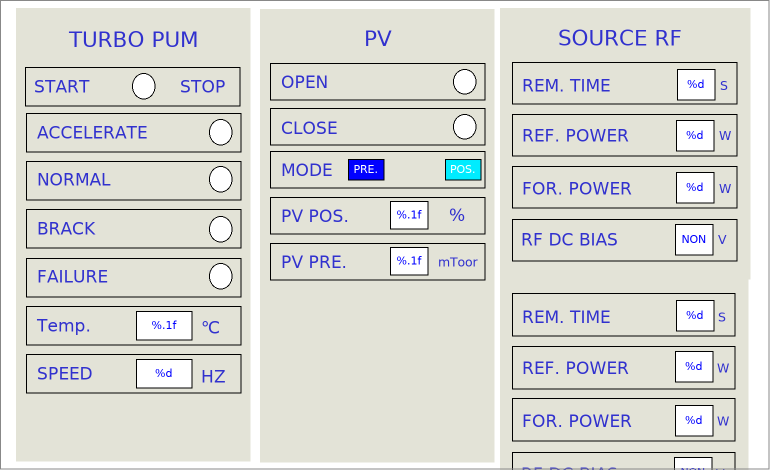
VISUALIZATION ViewPar  // 770x470
    RoundedRectangle (16,8 234x453)
    Label (38,17 192x45), "TURBO PUM"
    Ellipse (132,73 23x26), colour toggle: gICP.TruboPumOpen
    Label (31,75 67x23), "START"
    RoundedRectangle (26,113 215x39)
    RoundedRectangle (26,209 215x39)
    Ellipse (209,166 23x26), colour toggle: gICP.TruboPumNormal
    Label (34,168 117x23), "NORMAL"
    RoundedRectangle (26,161 215x39)
    Ellipse (209,119 23x26), colour toggle: gICP.TruboPumAcc
    Label (34,121 140x23), "ACCELERATE"
    RoundedRectangle (26,258 215x39)
    Ellipse (209,216 23x26), colour toggle: gICP.TruboPumDcc
    Label (34,217 117x23), "BRACK"
    RoundedRectangle (26,306 215x39)
    Ellipse (209,263 23x26), colour toggle: gICP.TruboPumError
    Label (34,265 117x23), "FAILURE"
    RoundedRectangle (26,354 215x39)
    Label (34,362 70x23), "SPEED"
    Label (198,365 31x23), "HZ"
    RoundedRectangle (136,359 56x29), "%d", text variable: gICP.TruboPumRotationSpeed
    Label (177,75 57x23), "STOP"
    Label (34,314 105x23), "Temp."
    Label (198,316 31x23), "℃"
    RoundedRectangle (136,311 56x29), "%.1f", text variable: gICP.TruboPumTMS
    RoundedRectangle (25,67 215x39)
    RoundedRectangle (260,9 234x453)
    Label (282,17 192x43), "PV"
    RoundedRectangle (270,63 215x37)
    Ellipse (453,69 23x25), colour toggle: gICP.PDVOpenSensor
    Label (278,71 117x22), "OPEN"
    RoundedRectangle (270,108 215x37)
    Ellipse (453,114 23x25), colour toggle: gICP.PDVCloseSensor
    Label (278,117 117x22), "CLOSE"
    RoundedRectangle (270,151 215x37)
    Label (278,159 69x22), "MODE"
    RoundedRectangle (270,197 215x37)
    Label (278,205 87x22), "PV POS."
    RoundedRectangle (270,243 215x37)
    Label (278,251 87x22), "PV PRE."
    RoundedRectangle (348,159 36x21), "PRE.", colour toggle: gICP.PDVModeRelay
    RoundedRectangle (445,159 36x21), "POS.", colour toggle: gICP.PDVModeRelay
    Label (446,204 23x22), "%"
    RoundedRectangle (390,201 38x28), "%.1f", text variable: gICP.PDV.actPos
    RoundedRectangle (390,247 38x28), "%.1f", text variable: gICP.PDV.actPressure
    Label (435,251 47x22), "mToor"
    Group (500,236 250x225)
        RoundedRectangle (0,0 248x276)
        Label (24,5 190x50), "POWER RF"
        RoundedRectangle (12,57 223x43)
        RoundedRectangle (12,110 223x43)
        RoundedRectangle (12,162 223x43)
        RoundedRectangle (12,216 223x43)
        Label (19,69 154x24), "REM. TIME"
        RoundedRectangle (176,64 38x31), "%d", text variable: gICP.PowerRF.rematime, colour toggle: gICP.PowerRF.rematime<>0
        Label (215,69 16x24), "S"
        Label (19,120 154x24), "REF. POWER"
        RoundedRectangle (175,115 38x31), "%d", text variable: gICP.PowerRF.reflectedpower, colour toggle: gICP.PowerRF.reflectedpower<>0
        Label (214,120 16x24), "W"
        Label (19,173 154x24), "FOR. POWER"
        RoundedRectangle (175,169 38x31), "%d", text variable: gICP.PowerRF.forwardpower, colour toggle: (gICP.PowerRF.openbusy AND ABS(gICP.PowerRF.forwardpower-gICP.PowerRF.setpower)>2) OR (not gICP.PowerRF.busy and gICP.PowerRF.forwardpower>0) OR (gICP.PowerRF.closebusy and gICP.PowerRF.forwardpower>0)
        Label (214,173 16x24), "W"
        Label (18,226 154x24), "RF DC BIAS"
        RoundedRectangle (174,221 38x31), "NON"
        Label (213,226 16x24), "V"
    Group (500,8 250x225)
        RoundedRectangle (0,0 250x271)
        Label (24,5 192x50), "SOURCE RF"
        RoundedRectangle (12,54 225x42)
        RoundedRectangle (12,106 225x42)
        RoundedRectangle (12,158 225x42)
        RoundedRectangle (12,211 225x42)
        Label (19,66 155x23), "REM. TIME"
        RoundedRectangle (177,61 38x31), "%d", text variable: gICP.SourceRF.rematime, colour toggle: gICP.SourceRF.rematime<>0
        Label (217,66 16x23), "S"
        Label (19,116 155x23), "REF. POWER"
        RoundedRectangle (176,112 38x31), "%d", text variable: gICP.SourceRF.reflectedpower, colour toggle: gICP.SourceRF.reflectedpower<>0
        Label (216,116 16x23), "W"
        Label (19,169 155x23), "FOR. POWER"
        RoundedRectangle (176,164 38x31), "%d", text variable: gICP.SourceRF.forwardpower, colour toggle: (gICP.SourceRF.busy AND ABS(gICP.SourceRF.forwardpower-gICP.SourceRF.setpower)>2) OR (not gICP.SourceRF.busy and gICP.SourceRF.forwardpower>0)
        Label (216,169 16x23), "W"
        Label (18,220 155x23), "RF DC BIAS"
        RoundedRectangle (175,216 38x31), "NON"
        Label (215,220 16x23), "V"
END_VISUALIZATION

(* stored: Version 1.1.0.1, ProductVersion 3.1.4024.12
   Visu ViewPar: Id {cba9ddf3-0a02-41b7-8579-e513daf9f3b5} *)
